// TIA Portal V20 export
TYPE "LKinCtrl_typeConfigurationKinematics"
   STRUCT
      "name" { ExternalAccessible := 'False'; ExternalVisible := 'False'; ExternalWritable := 'False'; S7_SetPoint := 'True'} : WString["LKINCTRL_LENGTH_OF_TO_NAME"];
      jogPath { ExternalAccessible := 'False'; ExternalVisible := 'False'; ExternalWritable := 'False'; S7_SetPoint := 'True'} : "LKinCtrl_typeJogConfiguration";
      jogOrientation { ExternalAccessible := 'False'; ExternalVisible := 'False'; ExternalWritable := 'False'; S7_SetPoint := 'True'} : "LKinCtrl_typeJogConfiguration";
   END_STRUCT;
   // jogPath.accelerationTime := 0.2;
   // jogPath.maxVelocityManual := 250.0;
   // jogPath.maxVelocityTestRun := 250.0;
   // jogPath.presetIncrementCoarse := 10.0;
   // jogPath.presetIncrementFine := 1.0;
   // jogPath.presetIncrementPrecise := 0.1;
   // jogOrientation.accelerationTime := 0.2;
   // jogOrientation.maxVelocityManual := 10.0;
   // jogOrientation.maxVelocityTestRun := 10.0;
   // jogOrientation.presetIncrementCoarse := 5.0;
   // jogOrientation.presetIncrementFine := 1.0;
   // jogOrientation.presetIncrementPrecise := 0.1;
END_TYPE
